//Check Error during FB_Init
IF THIS^.bErrorDuringFbInit THEN
	IF NOT fbInitError.bRaised THEN 
		//This error cannot be reset. Requires a reset cold
		fbInitError.CreateEx(stEventEntry:=TC_EVENTS.CHALET_Base_Events.ErrorFBinit, ipSourceInfo := THIS^.fbSourceInfo, bWithConfirmation := FALSE);
		fbInitError.Raise(0);
	END_IF
	Initialize:= E_FAIL;
	THIS^.fbFeedback.HR := Initialize;
	RETURN;
END_IF	

//Interface to System is missing
IF THIS^.ipXtsSystem = 0 THEN
	IF NOT fbMissingInterfaceAlarm.bRaised THEN 
		//This error cannot be reset. Requires a reset cold
		fbMissingInterfaceAlarm.CreateEx(stEventEntry:=TC_EVENTS.CHALET_XTS_Events.InitializationInvalideParameter, ipSourceInfo := THIS^.fbSourceInfo, bWithConfirmation := FALSE);
		fbMissingInterfaceAlarm.Raise(0);
	END_IF
	Initialize := E_FAIL;
	THIS^.fbFeedback.HR := Initialize;
	RETURN;
END_IF


IF NOT THIS^.bInitDone THEN
	
	THIS^.DeleteMoversQueue();

//	//Validate Settings - Error
//	bErrorStationInFrontNotFound := ((ipStationInFront = 0) AND THIS^.ipXtsSystem.Environment.TrackIsRing AND (THIS^.ipXtsSystem.Stations.Size > 1));
//	bErrorStationBehindeNotFound := ((ipStationBehinde = 0) AND THIS^.ipXtsSystem.Environment.TrackIsRing AND (THIS^.ipXtsSystem.Stations.Size > 1));		
//	IF (bErrorStationInFrontNotFound OR bErrorStationBehindeNotFound OR (THIS^.LUID = '') OR (fTrackLentgh <= 0) OR (fPositionOnTrack < 0.0) OR (fPositionOnTrack >= fTrackLentgh) OR (fMoverVelocityAtExit <= 0) OR (fMoverGapAtExit <= 0)) THEN
//		fbFeedback.hr := GetMostSignificant(E_FAIL, fbFeedback.hr);	
//		IF NOT fbInitError.bRaised THEN 
//			//This error cannot be reset. Requires a reset cold
//			fbInitError.CreateEx(stEventEntry:=TC_EVENTS.CHALET_XTS_Events.InitializationInvalideParameter, ipSourceInfo := THIS^.fbSourceInfo, bWithConfirmation := FALSE);
//			fbInitError.Raise(0);
//		END_IF
//	END_IF

		THIS^.fbTrigger.ListOfMoversToCheck := THIS^.ipXtsSystem.Movers;
		THIS^.fbTrigger.PositionOnTrack := THIS^.PositionOnTrack;
		THIS^.fbTrigger.TriggerDirection := MC_Positive_Direction;
		fbSortedListMoversInQueue.EndPositionOnTrack := LMOD(lr_Value:=(THIS^.PositionOnTrack + 10.0), lr_Arg:= THIS^.fTrackLentgh); 
		fbSortedListMoversInQueue.StartPositionOnTrack := LMOD(lr_Value:=(fbSortedListMoversInQueue.EndPositionOnTrack  + 0.0001), lr_Arg:= THIS^.fTrackLentgh); 
		fbSortedListMoversInQueue.ListOfMoversToCheck := THIS^.fbAssignedMovers;	
	bInitDone := TRUE;
END_IF

IF 	bInitDone THEN
	fbFeedback.hr := S_OK;	
END_IF
							
Initialize := fbFeedback.hr;
END_METHOD

{attribute 'monitoring':='call'}
//[mm] Every mover that leaves or passes the station gets this new gap as a target.
PROPERTY MoverGapAtExit : LREAL
GET
MoverGapAtExit := fMoverGapAtExit;
END_GET
SET
fMoverGapAtExit := MoverGapAtExit;
END_SET
END_PROPERTY

{attribute 'monitoring':='call'}
PROPERTY MoverPerMin : LREAL
GET
MoverPerMin := THIS^.fMoverPerMin;
END_GET
END_PROPERTY

{attribute 'monitoring':='call'}
PROPERTY MoverQueueSize : UINT
GET
MoverQueueSize := THIS^.nMoverQueueSize;
END_GET
SET
THIS^.nMoverQueueSize := MoverQueueSize;
END_SET
END_PROPERTY

{attribute 'monitoring':='call'}
PROPERTY MoversInPlace : BOOL
GET
THIS^.Prepare();//Prepare time-critical information, if not already done


MoversInPlace := bMoversInPlace;
END_GET
END_PROPERTY

{attribute 'monitoring':='call'}
PROPERTY MoversInQueue : REFERENCE TO ARRAY [0..(XtsParameterlist.MAX_MOVER_PER_SYSTEM-1)] OF I_XTS_Mover_PLC // Return a sorted list of movers in this zone. Index 0 is the mover in Front.
GET
MoversInQueue REF= THIS^.fbSortedListMoversInQueue.MoversInZone;
END_GET
END_PROPERTY

{attribute 'monitoring':='call'}
PROPERTY MoverVelocityAtExit : LREAL //[mm/s] Every mover that leaves or passes the station gets this new velocity as a target.
GET
MoverVelocityAtExit := fMoverVelocityAtExit;
END_GET
SET
fMoverVelocityAtExit := MoverVelocityAtExit;
END_SET
END_PROPERTY

PROPERTY OID : OTCID
GET
OID := THIS^.OIDStationInfo;
END_GET
END_PROPERTY

{attribute 'monitoring':='call'}
//[mm] from the beginning of the assigned track
PROPERTY PositionOnTrack : LREAL
GET
PositionOnTrack := fPositionOnTrack;
END_GET
SET
THIS^.ChangePos(PositionOnTrack);
END_SET
END_PROPERTY

(* 
	Use this Methode to calculate time sensitive date once each cycle. Example: read analog input and convert before do get Signal propertie
*)
METHOD PROTECTED Prepare : HRESULT
VAR_INST
	{attribute 'hide'}	
	nLastUpdatedCycleCount : UDINT;
END_VAR

VAR
	nLoopIndex : UINT;
	fExpectedDistanceToParent : LREAL;
	fPositionDifference : LREAL;
	nCycleTime_ms : UDINT;
	bMoverInQueue : BOOL;
	bTempMoverInPosition : BOOL;
	bTempMoverVeloZero : BOOL;
	bTempMoverInMonitoringTime : BOOL;
	bTempMoverThisStationAsTarged : BOOL;
END_VAR
VAR_INST
	{attribute 'hide'}
	nCycleCountInPos : UDINT;
END_VAR
//Check if this Cycle the dates are allready prepared. This is important for time sensitive informations.
IF nLastUpdatedCycleCount <> TwinCAT_SystemInfoVarList._TaskInfo[THIS^.TaskIndex].CycleCount THEN
	nLastUpdatedCycleCount := TwinCAT_SystemInfoVarList._TaskInfo[THIS^.TaskIndex].CycleCount ;


	(* Check if mover is in place. Time and Position window *)
	//If queuesize is zero, mover is never in place.
	IF nMoverQueueSize = 0 OR NOT ipXtsSystem.Enabled THEN
		THIS^.bMoversInPlace := FALSE;
		nCycleCountInPos := 0;
	ELSE
		//Get this task cycle Count and time 
		nCycleTime_ms := TwinCAT_SystemInfoVarList._TaskInfo[THIS^.nTaskIndex].CycleTime(*100ns*) / 10_000 ;
		
		bTempMoverInPosition := TRUE; bTempMoverVeloZero := TRUE; bTempMoverThisStationAsTarged := TRUE;
		fExpectedDistanceToParent := 0;
		FOR nLoopIndex := 0 TO (THIS^.nMoverQueueSize-1) DO
			IF THIS^.fbSortedListMoversInQueue.MoversInZone[nLoopIndex] <> 0 THEN
				//Check position and Gap - 1 mover do not have a gap
				IF nLoopIndex <> 0 THEN
					fExpectedDistanceToParent := fExpectedDistanceToParent + THIS^.fbSortedListMoversInQueue.MoversInZone[nLoopIndex].LastCmdTargedGap;
				END_IF
				bMoverInQueue		:= TRUE;
				
				fPositionDifference := F_GetDistToPosModulo(fTargedPosition := (THIS^.PositionOnTrack - fExpectedDistanceToParent),  fActualPosition :=  THIS^.fbSortedListMoversInQueue.MoversInZone[nLoopIndex].FullAccess.getAxisRef.NcToPlc.ModuloActPos, fModulo := THIS^.ipXtsSystem.TrackLength);
				IF fPositionDifference > (THIS^.ipXtsSystem.TrackLength/2) THEN
					fPositionDifference := (THIS^.ipXtsSystem.TrackLength - fPositionDifference);
				END_IF
				
				bTempMoverInPosition := bTempMoverInPosition AND (ABS(fPositionDifference) <= fTargetPosWindow );
				bTempMoverVeloZero := bTempMoverVeloZero AND (THIS^.fbSortedListMoversInQueue.MoversInZone[nLoopIndex].SetVelocity = 0);
				bTempMoverThisStationAsTarged := bTempMoverThisStationAsTarged AND ((THIS^.fbSortedListMoversInQueue.MoversInZone[nLoopIndex].TargedStation = THIS^.LUID));
			ELSE
				//Missing mover in queue
				bMoverInQueue := FALSE;
				EXIT;
			END_IF
		END_FOR
			
		//start time if mover position is ok
		IF bTempMoverInPosition  THEN
			nCycleCountInPos := nCycleCountInPos + 1;
		ELSE
			nCycleCountInPos := 0;
		END_IF
		
		bTempMoverInMonitoringTime := (UDINT_TO_TIME(nCycleCountInPos * nCycleTime_ms) >= tTargetPosMonitoringTime);
				
		THIS^.bMoversInPlace := bMoverInQueue AND bTempMoverInPosition AND bTempMoverInMonitoringTime AND bTempMoverThisStationAsTarged;// AND bTempMoverVeloZero;
	END_IF
	
	
END_IF
END_METHOD

{attribute 'monitoring':='call'}
PROPERTY ProcessSimulationActive : BOOL
GET
ProcessSimulationActive := THIS^.fSimulationProcessDuration > 0;
END_GET
END_PROPERTY

{attribute 'monitoring':='call'}
//prevent further movers from entering the station, 
//e.g. to prevent a collision. All movers that are already moving to reach this station will be stopped with a stop 
//and restarted with Ready True.
PROPERTY ReadyToRecvMovers : BOOL
GET
ReadyToRecvMovers := bReadyToRecvMovers;
END_GET
SET
VAR
	ipTempMover : I_XTS_Mover;
END_VAR
//Change to Not Ready:
IF (ReadyToRecvMovers = FALSE) AND (bReadyToRecvMovers <> ReadyToRecvMovers) THEN
	//halt all movers on the way
	fbAssignedMovers.ResetIterator();
	WHILE fbAssignedMovers.HasNextObject() DO
		IF ToMover(fbAssignedMovers.GetNextObject(),ipTempMover) THEN
			ipTempMover.HaltCA();	
		END_IF	
	END_WHILE
END_IF

//Change to Ready:
IF (ReadyToRecvMovers = TRUE) AND (bReadyToRecvMovers <> ReadyToRecvMovers) THEN
	//all movers that are on the way have probably been stopped before. when reactivated, the last move command is sent again.
	fbAssignedMovers.ResetIterator();
	WHILE fbAssignedMovers.HasNextObject() DO
		IF ToMover(fbAssignedMovers.GetNextObject(),ipTempMover) THEN
			ipTempMover.MoveAbsCA(	fPosition	:= THIS^.PositionOnTrack, 
								fVelocity 	:= ipTempMover.LastCmdTargedVelocity,  
								fGap 		:= ipTempMover.LastCmdTargedGap,  
								eDirection 	:= Tc3_Mc3Definitions.MC_DIRECTION.mcDirectionPositive);	
		END_IF	
	END_WHILE
END_IF

//Store new status
bReadyToRecvMovers := ReadyToRecvMovers;
END_SET
END_PROPERTY

METHOD SendMoversToStation : HRESULT //Send all Queued movers away by changing the targed station destination
VAR_INPUT
	sTargedStation	: STRING;
END_VAR
VAR
	nLoopIndex 		: UINT;;
	ipMover	: I_XTS_Mover;
END_VAR
//Invalide targed
IF sTargedStation = '' THEN
	SendMoversToStation := E_FAIL;
	RETURN;
END_IF

//Movers have not reached station and can not send away until complet
IF NOT THIS^.MoversInPlace THEN
	SendMoversToStation := E_FAIL;
	RETURN;
END_IF

//Send all Queued movers away by changing the targed station destination
FOR nLoopIndex := 0 TO nMoverQueueSize-1 DO
	IF THIS^.MoversInQueue[nLoopIndex] <> 0 AND_THEN __QUERYINTERFACE(THIS^.MoversInQueue[nLoopIndex],ipMover) THEN
		ipMover.TargedStation := sTargedStation;		
	END_IF
END_FOR
END_METHOD

//If a valid time (>0seconds) is set and the configured destination station exists, then the movers will be sent away automatically after this time from now on.
METHOD SimulationStart : HRESULT
VAR_INPUT
	fProcessDuration 	: LREAL; //[s]
	sTargedStation		: STRING; //LUID of the targed station to automatic send after the duration
END_VAR
VAR
	ipStation	: I_CH_Object;
	bValideLUID : BOOL;
END_VAR
//Search LUID in Stationslist
ipStation := THIS^.ipXtsSystem.Stations.FindLUID(sTargedStation);
bValideLUID := (ipStation <> 0); 

IF (fProcessDuration > 0) AND bValideLUID THEN
	//Valide config
	THIS^.fSimulationProcessDuration 	:=	fProcessDuration;
	THIS^.sSimulationTargedStation 		:=	sTargedStation;
	SimulationStart := S_OK;
ELSE
	//Simulation disabled
	THIS^.SimulationStop();
	SimulationStart := S_FALSE;
END_IF
END_METHOD

//If a valid time (>0seconds) is set and the configured destination station exists, then the movers will be sent away automatically after this time from now on.
METHOD SimulationStartEx : HRESULT
VAR_INPUT
	fProcessDuration 		: LREAL; //[s]
	ipStation				: I_Xts_Station_PLC; //unique station to automatic send after the duration
END_VAR
IF ipStation <> 0 THEN
	SimulationStartEx := THIS^.SimulationStart(fProcessDuration := fProcessDuration, sTargedStation := ipStation.LUID);

ELSE
	SimulationStartEx := S_FALSE;
END_IF
END_METHOD

METHOD SimulationStop : HRESULT
//Simulation disabled
THIS^.fSimulationProcessDuration 	:=	0;
THIS^.sSimulationTargedStation 		:=	'';
END_METHOD

{attribute 'monitoring':='call'}
PROPERTY StationBehinde : I_XTS_Station
GET
StationBehinde := ipStationBehinde;
END_GET
END_PROPERTY

{attribute 'monitoring':='call'}
PROPERTY StationsAhead : I_XTS_Station
GET
StationsAhead := ipStationInFront;
END_GET
END_PROPERTY

{attribute 'monitoring':='call'}
PROPERTY SuppressDynamicsChange : BOOL // Suppress to change the dynamic(Gap+velocity) of passing movers. This is usefull in startup
GET
SuppressDynamicsChange := bSuppressDynamicsChange;
END_GET
SET
bSuppressDynamicsChange := SuppressDynamicsChange;
END_SET
END_PROPERTY

{attribute 'monitoring':='call'}
//A time that is waited as soon as the mover is in the station (including the monitoring window) before “MoversInPlace” is set. e.g. used to stabilize the workpiece
PROPERTY TargetPosMonitoringTime : TIME
GET
TargetPosMonitoringTime := tTargetPosMonitoringTime;
END_GET
SET
tTargetPosMonitoringTime := TargetPosMonitoringTime;
END_SET
END_PROPERTY

{attribute 'monitoring':='call'}
//How many mm before the mover reaches the position is “MoversInPlace” set for the process. 
//This distance can also be set very large (e.g. 100mm) for moving past without stopping.
PROPERTY TargetPosWindow : LREAL
GET
TargetPosWindow := fTargetPosWindow;
END_GET
SET
fTargetPosWindow := TargetPosWindow;
END_SET
END_PROPERTY

//This sequence tries to transfer the mover to the next station in the direction of travel and checks whether the next station has space for it. 
//If the next station is a "dummy" that only changes the dynamics of the passing mover, this station is skipped and the next station is searched one ahead.
//If the station is fully occupied, no action is taken and a new search can be made in the next cycle.
METHOD PROTECTED TrySendMoverToNextStation : HRESULT
VAR_INPUT
	ipMover	: I_XTS_Mover;
	fVelocity : LREAL;
	fGap : LREAL;
END_VAR
VAR
	bStationIsOnlyForDynamicChanges : BOOL;
	bStationIsFull					: BOOL;
	bStationHanMoreMoverThanAllowed : BOOL;
	bStationHasAFreePlaceInQueue 	: BOOL;
	bStationIsTheTarged				: BOOL;
	bStationIsNotReadyToRecvMovers	: BOOL;
	
	ipMoverObject 		: I_CH_Object;
	ipTempStation 		: I_XTS_Station;	
	ipTargedStation 	: I_XTS_Station;

	nXpuNo 				: UINT;
	iMoverNo 			: UINT;
	stCommand 			: ST_TcIoXtsMoverCommand;	
END_VAR
//Invalide interface
IF ipMover = 0 THEN
	TrySendMoverToNextStation := E_FAIL;
	RETURN;
END_IF

//Mover is not in this Station.
IF __QUERYINTERFACE(ipMover,ipMoverObject) AND_THEN NOT THIS^.fbAssignedMovers.ObjectInList(ipMoverObject) THEN
	TrySendMoverToNextStation := E_FAIL;
	RETURN;
END_IF

//Send to actual Station is not supported
IF ipMover.TargedStation = THIS^.LUID THEN
	TrySendMoverToNextStation := E_FAIL;
	RETURN;
END_IF


ipTempStation := (THIS^);
//This sequence tries to transfer the mover to the next station in the direction of travel and checks whether the next station has space for it. 
//If the next station is a "dummy" that only changes the dynamics of the passing mover, this station is skipped and the next station is searched one ahead.
//If the station is fully occupied, no action is taken and a new search can be made in the next cycle.
WHILE (ipTargedStation=0) DO
	
	//get next station in flow direction
	ipTempStation := ipTempStation.StationsAhead;

	//All Stations around the XTS tested, Station not Found
	IF ipTempStation.LUID = THIS^.LUID THEN
		TrySendMoverToNextStation := E_FAIL;
		RETURN;
	END_IF

	bStationHanMoreMoverThanAllowed := (ipTempStation.CtsMoversInQueue > ipTempStation.MoverQueueSize); //Maybe during statup if all movers are forced to station x.	
	bStationIsFull					:= (ipTempStation.CtsEmptySpaceInQueue = 0) AND NOT (ipTempStation.MoverQueueSize = 0);
	bStationHasAFreePlaceInQueue 	:= (ipTempStation.CtsEmptySpaceInQueue > 0);
	bStationIsOnlyForDynamicChanges := (ipTempStation.MoverQueueSize = 0);
	bStationIsTheTarged				:= (ipTempStation.LUID = ipMover.TargedStation);
	bStationIsNotReadyToRecvMovers	:= ( NOT ipTempStation.ReadyToRecvMovers); 
	
	IF bStationIsFull OR bStationHanMoreMoverThanAllowed OR bStationIsNotReadyToRecvMovers THEN
		//Next Station is a valide targed but is already full.  Exit WHILE loop and try again next time.
		EXIT;
	
	ELSIF bStationHasAFreePlaceInQueue THEN
		//Next station found. Send mover to it.
		ipTargedStation := ipTempStation;
	
	ELSIF bStationIsOnlyForDynamicChanges AND bStationIsTheTarged THEN
		//ERROR. The target position is a dynamic station and can not be reached.
		TrySendMoverToNextStation := E_FAIL;
		RETURN;
		
	ELSIF bStationIsOnlyForDynamicChanges THEN
		//Repead WHILE loop and search an station more in front.
		;
	END_IF 

END_WHILE


//Requested station was found, send movers to there if it has space.
IF ipTargedStation <> 0 THEN
	//Handover Mover
	THIS^.fbAssignedMovers.RemoveObject(ipMoverObject);
	ipTargedStation.AddMoverToQueue(ipMover);
	//Start Movement
	ipMover.MoveAbsCA(
		fPosition:= ipTargedStation.PositionOnTrack, 
		fVelocity:= fVelocity, 
		fGap:= fGap, 
		eDirection:= Tc3_Mc3Definitions.MC_DIRECTION.mcDirectionPositive);
		
	//build Log Command
	stCommand.sCommandType	:= 'leaving station';
	stCommand.sStation		:= ipTargedStation.LUID;
	stCommand.sText 		:= F_BuildLogString(fPos := ipTargedStation.PositionOnTrack, fVelocity := fVelocity, fGap := fGap);

	//get Xpu Number by AxisId
	nXpuNo := ipXtsSystem.Environment.UtilityEnvirement.GetXpuNumberByAxisId(ipMover.getAxisRef.NcToPlc.AxisId);
	//get Mover Number by AxisId
	iMoverNo := ipXtsSystem.Environment.UtilityEnvirement.XpuTcIo(nXpuNo).GetMoverNumberByAxisId(ipMover.getAxisRef.NcToPlc.AxisId);
	
	//write Log Command
	ipXtsSystem.Environment.UtilityEnvirement.XpuTcIo(nXpuNo).MoverTcIo(iMoverNo).AddCommand(stCommand);
	

	
	TrySendMoverToNextStation := S_OK;	
ELSE
	//No movemnt possible, try next cycle again		
	TrySendMoverToNextStation := S_FALSE;
END_IF
END_METHOD

METHOD Update : HRESULT
VAR
	ipMover : I_XTS_Mover;
	ipThisStation : I_XTS_Station;
	fDistToNextMover : LREAL;
	fGapRequired : LREAL;
	bGapIsEnough : BOOL; //distance is large enough to start next command
END_VAR
//Force to do init befor call update
IF NOT bInitDone THEN
	THIS^.Initialize();
	RETURN;
END_IF


// Process Simulation. All functionality packed into one method for easier overwriting
THIS^.UpdateSimulation();


// If enabled start station logic
IF THIS^.ipXtsSystem.Enabled THEN
	
	ipThisStation := (THIS^);
	//Detect mover who is passing the station whitout be in queue. Adjust to new Gap+Dynamics
	IF fbTrigger.MoverDetected AND fbTrigger.MoverAtTrigger<>0 AND NOT THIS^.bSuppressDynamicsChange THEN
		//Only if not in this queue
		IF fbTrigger.MoverAtTrigger.ParentStation <> ipThisStation THEN
			fbTrigger.MoverAtTrigger.MoveAbsCA(
				fPosition:= fbTrigger.MoverAtTrigger.LastCmdTargedPosition, 
				fVelocity:= THIS^.fMoverVelocityAtExit, 
				fGap:= THIS^.fMoverGapAtExit, 
				eDirection:= Tc3_Mc3Definitions.MC_DIRECTION.mcDirectionPositive);
		END_IF
	END_IF
	
	///distance is large enough to start next command
	//This is to prevent stationary movers from having to move backwards
	IF THIS^.MoversInQueue[0] <> 0 THEN
		fDistToNextMover := F_GetDistToPosModulo(fTargedPosition:= THIS^.MoversInQueue[0].FullAccess.NextMover.PositionOnTrack, fActualPosition:= THIS^.MoversInQueue[0].PositionOnTrack, THIS^.ipXtsSystem.TrackLength);
		fGapRequired := MAX(THIS^.MoversInQueue[0].FullAccess.LastCmdTargedGap, THIS^.MoversInQueue[0].FullAccess.NextMover.LastCmdTargedGap);
		bGapIsEnough := (fDistToNextMover >= fGapRequired);
	END_IF
	
	
	//Test if the first mover is in station and send him away, if the destination is not this station
	IF __QUERYINTERFACE(THIS^.MoversInQueue[0],ipMover) AND_THEN (ipMover.TargedStation <> THIS^.LUID) AND_THEN bGapIsEnough THEN
		//IF mover is standstill in current station, send him away whit the exitVelocity, else use the in mover stored velocity
		IF (THIS^.MoversInQueue[0].PositionOnTrack = THIS^.PositionOnTrack) THEN
			THIS^.TrySendMoverToNextStation(ipMover := ipMover, fVelocity := THIS^.fMoverVelocityAtExit, fGap := THIS^.fMoverGapAtExit);
		ELSE
			THIS^.TrySendMoverToNextStation(ipMover := ipMover, fVelocity := ipMover.LastCmdTargedVelocity, fGap := ipMover.LastCmdTargedGap);
		END_IF	
      
	END_IF
END_IF


// Utility InfoStation, used in XTS Viewer. All functionality packed into one method for easier overwriting
THIS^.UpdateUtilityStation();

// Calculate statistic values like Mover/min of this station. All functionality packed into one method for easier overwriting
THIS^.UpdateStatistic();
END_METHOD

METHOD PROTECTED UpdateSimulation : HRESULT
VAR_INST
	tonSimulationDelay : TON;
END_VAR
//Automatic send mover to next station in Simulation
//If a valid time (>0seconds) is set and the configured destination station exists, then the movers will be sent away automatically after this time from now on.
tonSimulationDelay.IN 	:= THIS^.ipXtsSystem.Enabled AND THIS^.MoversInPlace AND THIS^.ProcessSimulationActive;
tonSimulationDelay.PT	:= LREAL_TO_TIME(THIS^.fSimulationProcessDuration*1000.0);
tonSimulationDelay();
IF tonSimulationDelay.Q THEN
	THIS^.SendMoversToStation(sTargedStation := THIS^.sSimulationTargedStation);
END_IF
END_METHOD

METHOD PROTECTED UpdateStatistic : HRESULT
VAR
	nCycleTime_ns : UDINT;
END_VAR
VAR_INST
	tWaitForXTS, tWaitForProcess 	: LTIME;
	nMoverPassingStation			: UINT;
END_VAR
//Validate settings. STATISTIC_AVG_PERIOD must be >0
IF NOT TIME_TO_BOOL(XtsParameterlist.STATISTIC_AVG_PERIOD) THEN
	UpdateStatistic := E_FAIL;
	RETURN;
END_IF

//Get this task cycle time
nCycleTime_ns := TwinCAT_SystemInfoVarList._TaskInfo[THIS^.nTaskIndex].CycleTime(*100ns*) * 100;


//Depending on whether the station gives the start signal to the process or not, decide which of the two times should be incremented.
IF THIS^.MoversInPlace THEN
	tWaitForProcess := tWaitForProcess + UDINT_TO_LTIME(nCycleTime_ns);
ELSE
	tWaitForXTS 	:= tWaitForXTS + UDINT_TO_LTIME(nCycleTime_ns);
END_IF


//Check for mover who is passing the station
IF THIS^.fbTrigger.MoverDetected THEN
	nMoverPassingStation := nMoverPassingStation +1;
END_IF


//Once the period is reached. Evaluate and reset
IF (tWaitForProcess + tWaitForXTS) >= TIME_TO_LTIME(XtsParameterlist.STATISTIC_AVG_PERIOD) THEN
	
	//Calculate passing mover per minute
	THIS^.fMoverPerMin := TO_LREAL(nMoverPassingStation)*TIME_TO_LREAL(TIME#1M)/TIME_TO_LREAL(XtsParameterlist.STATISTIC_AVG_PERIOD);

	
	
	tWaitForProcess	:= LTIME#0NS;
	tWaitForXTS 	:= LTIME#0NS;
	nMoverPassingStation := 0;
END_IF
END_METHOD

METHOD PROTECTED UpdateUtilityStation : HRESULT //Utility InfoStation, used in XTS Viewer. All functionality packed into one method for easier overwriting
VAR
	aStopPositionsInfoStation : ARRAY[1..Tc3_XTS_Utility.TcIoXtsEnvironmentParameterList.MaxXtsStopPositionsPerStation] OF LREAL;
	//aPartIDs : ARRAY[1..Tc3_XTS_Utility.TcIoXtsEnvironmentParameterList.MaxXtsPartsPerXpu] OF OTCID;
	fLastStopPosition 		: LREAL;
	nLoopIndex 				: UINT;	
    ipMovers 				: CHALET_BaseComponents.I_CH_List;
	ipTempMover 			: I_XTS_Mover;
	nXpuNo 					: UINT;
	nMoverNo 				: UINT;
	pObject 				: ITComObject;
	sName 					: STRING;
END_VAR


VAR_INST

	nOldMoverQueueSize 		: UINT := CHALET_BaseComponents.GVL_Datatypes.cMaxUint;
	fOldPositionOnTrack 	: LREAL;
	anBias 					: ARRAY[1..2] OF INT;
	bInverted 				: BOOL;
END_VAR
//Validate inputs
IF THIS^.OIDStationInfo = 0 OR ipXtsSystem.Environment = 0 THEN
	RETURN;
END_IF	


// Initalize
IF NOT THIS^.bUtilityStationInitDone THEN
	//Get interface to utility station belongs to this station via OID
    FOR nLoopIndex := 1 TO ipXtsSystem.Environment.UtilityEnvirement.InfoServerTcIo(1).P_InfoStationCount DO
		IF 	ipXtsSystem.Environment.UtilityEnvirement.InfoServerTcIo(1).P_InfoStationOids[nLoopIndex] = THIS^.OIDStationInfo THEN
			THIS^.ipStationInfo := ipXtsSystem.Environment.UtilityEnvirement.InfoServerTcIo(1).InfoStationTcIo(nInfoStation:= nLoopIndex);
			EXIT;
		END_IF
	END_FOR	
	
	// calculate Position Offset
	IF THIS^.ipStationInfo <> 0 THEN			
		ipMovers := ipXtsSystem.Movers;
		ipMovers.ResetIterator();
		nLoopIndex := 0;	
		WHILE ipMovers.HasNextObject() DO
			nLoopIndex := nLoopIndex + 1;
			IF ToMover(ipMovers.GetNextObject(),ipTempMover) THEN
				//get Xpu Number by AxisId
				nXpuNo := ipXtsSystem.Environment.UtilityEnvirement.GetXpuNumberByAxisId(ipTempMover.getAxisRef.NcToPlc.AxisId);
				//get Mover Number by AxisId
				nMoverNo := ipXtsSystem.Environment.UtilityEnvirement.XpuTcIo(nXpuNo).GetMoverNumberByAxisId(ipTempMover.getAxisRef.NcToPlc.AxisId);
				//calculate Bias
				anBias[nLoopIndex] := LREAL_TO_INT(ipXtsSystem.Environment.UtilityEnvirement.XpuTcIo(nXpuNo).MoverTcIo(nMoverNo).GetPositionInfo().fPartPosition - ipTempMover.getAxisRef.NcToPlc.ModuloActPos);
				IF nLoopIndex = 2 THEN
					 EXIT;
				END_IF
			END_IF
		END_WHILE
		
		// Validate bias, check for inverted direction
		IF anBias[1] <> anBias[2] THEN
			bInverted := TRUE; 
			ipMovers.ResetIterator();
			nLoopIndex := 0;	
			WHILE ipMovers.HasNextObject() DO
				nLoopIndex := nLoopIndex + 1;
				IF ToMover(ipMovers.GetNextObject(),ipTempMover) THEN
					//get Xpu Number by AxisId
					nXpuNo := ipXtsSystem.Environment.UtilityEnvirement.GetXpuNumberByAxisId(ipTempMover.getAxisRef.NcToPlc.AxisId);
					//get Mover Number by AxisId
					nMoverNo := ipXtsSystem.Environment.UtilityEnvirement.XpuTcIo(nXpuNo).GetMoverNumberByAxisId(ipTempMover.getAxisRef.NcToPlc.AxisId);
					//calculate inverted Bias
					anBias[nLoopIndex] := LREAL_TO_INT(ipXtsSystem.TrackLength - ipXtsSystem.Environment.UtilityEnvirement.XpuTcIo(nXpuNo).MoverTcIo(nMoverNo).GetPositionInfo().fPartPosition - ipTempMover.getAxisRef.NcToPlc.ModuloActPos);
					IF nLoopIndex = 2 THEN
						 EXIT;
					END_IF
				END_IF	
			END_WHILE
		END_IF
		
		//Set unique station name
		FW_ObjMgr_GetObjectInstance(oid:= THIS^.OIDStationInfo , iid:= TC_GLOBAL_IID_LIST.IID_ITComObject, pipUnk:= ADR(pObject));
		IF pObject <> 0 THEN
			sName := THIS^.LUID;
			pObject.TcSetObjectName(ADR(sName));
			pObject.TcRelease();
		END_IF

	END_IF
	
	THIS^.bUtilityStationInitDone := TRUE;
	fOldPositionOnTrack := -1;
END_IF




// Update
// Configure/draw station in viewer on change
IF (THIS^.ipStationInfo <> 0) AND (THIS^.nMoverQueueSize <> nOldMoverQueueSize OR THIS^.fPositionOnTrack <> fOldPositionOnTrack) THEN	
	nOldMoverQueueSize := THIS^.nMoverQueueSize;
	fOldPositionOnTrack := THIS^.fPositionOnTrack;
	
	THIS^.ipStationInfo.SetPartObjectIds(ipXtsSystem.Environment.UtilityEnvirement.XpuTcIo(1).P_PartOids);
	THIS^.ipStationInfo.SetIsEnabled(TRUE);

	
	// Draw stop position if gap between mover, given by station behind, is set
	IF (StationBehinde <> 0) AND (THIS^.nMoverQueueSize > 0) AND THIS^.nMoverQueueSize <= 25 THEN
		//Clear array
		MEMSET(ADR(aStopPositionsInfoStation), SIZEOF(aStopPositionsInfoStation), 0);
		//Fill array
		FOR nLoopIndex := 1 TO THIS^.nMoverQueueSize DO
			fLastStopPosition := (nLoopIndex-1)*StationBehinde.MoverGapAtExit;
			aStopPositionsInfoStation[(nLoopIndex)] := (fLastStopPosition);
		END_FOR
		IF NOT bInverted THEN
			//Start Position
			THIS^.ipStationInfo.SetStartPositionOnPart(MAX((fPositionOnTrack + anBias[1] - fLastStopPosition), 0)); ///zzz Todo. The InfoStation can not draw stations in the modulo area
			//End Pos
			THIS^.ipStationInfo.SetEndPositionOnPart(fPositionOnTrack + anBias[1]);
		ELSE
			//Start Position
			THIS^.ipStationInfo.SetStartPositionOnPart(ipXtsSystem.TrackLength - (fPositionOnTrack + anBias[1]));					
			//End Pos
			THIS^.ipStationInfo.SetEndPositionOnPart(MAX((ipXtsSystem.TrackLength - (fPositionOnTrack + anBias[1] - fLastStopPosition)), 0)); ///zzz Todo. The InfoStation can not draw stations in the modulo area
		END_IF
		//StopPositions
		THIS^.ipStationInfo.SetStopPositions(aStopPositionsInfoStation);

		//Override color if is set to transparent
		IF THIS^.ipStationInfo.GetStationColor() = 0 THEN
			THIS^.ipStationInfo.SetStationColor(nStationColor:= CHALET_BaseComponents.E_Colors_ARGB.Darkred);
		END_IF
	ELSE
		//Clear array
		MEMSET(ADR(aStopPositionsInfoStation), SIZEOF(aStopPositionsInfoStation), 0);	
		//StopPositions
		THIS^.ipStationInfo.SetStopPositions(aStopPositionsInfoStation);
		//Start Pos
		THIS^.ipStationInfo.SetStartPositionOnPart(nStartPositionOnPart := fPositionOnTrack + anBias[1]);
		//End Position
		THIS^.ipStationInfo.SetEndPositionOnPart(nEndPositionOnPart := fPositionOnTrack + anBias[1]);
	END_IF
	
	
	
	//Color Station depending on function:
	// Waitingstation green
	IF (FIND(THIS^.LUID,'wait')>0) OR (FIND(THIS^.LUID,'Wait')>0) OR (FIND(THIS^.LUID,'Warte')>0) OR (FIND(THIS^.LUID,'warte')>0) THEN
		THIS^.UtilityStationInfo.SetStationColor(nStationColor := CHALET_BaseComponents.E_Colors_ARGB.Green);
	
	// Dynamicstation blue
	ELSIF THIS^.MoverQueueSize = 0 THEN
		THIS^.UtilityStationInfo.SetStationColor(nStationColor := CHALET_BaseComponents.E_Colors_ARGB.Royalblue);	
    
	// Process station red
	ELSE
		THIS^.UtilityStationInfo.SetStationColor(nStationColor := CHALET_BaseComponents.E_Colors_ARGB.Red);			
	END_IF

END_IF
END_METHOD

{attribute 'monitoring':='call'}
PROPERTY UtilityStationInfo : I_TcIoXtsInfoServerInfoStation
GET
UtilityStationInfo := THIS^.ipStationInfo;
END_GET
END_PROPERTY

END_FUNCTION_BLOCK

// ---- COMPENENTs/Trigger/FB_XTS_Trigger.TcPOU
{attribute 'no_explicit_call' := 'Do not call the body - Stick to OOP'}
FUNCTION_BLOCK FB_XTS_Trigger EXTENDS FB_CH_Object IMPLEMENTS I_XTS_Trigger
VAR
	{attribute 'hide'}
	bInitDone : BOOL;
	{attribute 'hide'}
	ipXtsSystem : I_XTS_System_Registration;
	{attribute 'hide'}
	ipListOfMoversToCheck : CHALET_BaseComponents.I_CH_LIST;
	{attribute 'hide'}
	fTriggerPositionOnTrack : LREAL;
	{attribute 'hide'}
	eTriggerDirection : Tc2_MC2.MC_Direction := MC_Positive_Direction;
	{attribute 'hide'}
	ipMoverAtTrigger : I_XTS_Mover;
	{attribute 'hide'}	
	fTrackLentgh : LREAL;
	{attribute 'hide'}
	aMoversPositionLastCycle : ARRAY [0..(XtsParameterlist.MAX_MOVER_PER_SYSTEM-1)] OF LREAL; // This list is generated at the end of the PRG and contais the positions. The positions are checked in the next cycle
	{attribute 'hide'}
	aMoversInterfaceLastCycle : ARRAY [0..(XtsParameterlist.MAX_MOVER_PER_SYSTEM-1)] OF I_XTS_Mover; // This list is generated at the end of the PRG and contais the Mover interface. The positions are checked in the next cycle
	
END_VAR

METHOD FB_init : BOOL
VAR_INPUT
	bInitRetains : BOOL; // if TRUE, the retain variables are initialized (warm start / cold start)
	bInCopyCode : BOOL;  // if TRUE, the instance afterwards gets moved into the copy code (online change)
	
	ipXtsSystem : I_XTS_System_Registration; //Interface to XTS system object
	
END_VAR
VAR_INST
	{attribute 'hide'}
	bFBInitCalledOnce : BOOL; //Do the following code once during start up and not during onlinechange
END_VAR
//Do the following code once during start up and not during onlinechange
IF NOT bFBInitCalledOnce THEN 
	;
END_IF

//Regristrate object in System if unknown
IF ipXtsSystem <> 0 AND THIS^.ipXtsSystem = 0 THEN
	ipXtsSystem.RegisterTrigger(THIS^);
	THIS^.ipXtsSystem := ipXtsSystem;
END_IF

bFBInitCalledOnce := TRUE;
END_METHOD

{attribute 'monitoring':='call'}
PROPERTY HR : HRESULT
GET
///zzz todo
END_GET
END_PROPERTY

METHOD Initialize : HRESULT
IF THIS^.ipXtsSystem = 0 THEN
	//No valide interface
	Initialize := E_FAIL;
	RETURN;
END_IF

//Store track information
THIS^.fTrackLentgh := THIS^.ipXtsSystem.TrackLength;

IF (THIS^.ipListOfMoversToCheck <> 0) AND (THIS^.fTrackLentgh > 0.0) THEN
	THIS^.bInitDone := TRUE;
	Initialize := S_OK;
ELSE
	Initialize := E_FAIL;
END_IF
END_METHOD

PROPERTY ListOfMoversToCheck : I_CH_List
SET
IF ListOfMoversToCheck <> 0 THEN
	ipListOfMoversToCheck := ListOfMoversToCheck;
END_IF
END_SET
END_PROPERTY

{attribute 'monitoring':='call'}
PROPERTY MoverAtTrigger : I_XTS_Mover
GET
THIS^.Prepare();//Prepare Time-critical information

MoverAtTrigger := ipMoverAtTrigger;
END_GET
END_PROPERTY

{attribute 'monitoring':='call'}
PROPERTY MoverDetected : BOOL
GET
THIS^.Prepare();//Prepare Time-critical information

MoverDetected := (ipMoverAtTrigger <> 0);
END_GET
END_PROPERTY

{attribute 'monitoring':='call'}
PROPERTY PositionOnTrack : LREAL
GET
PositionOnTrack := fTriggerPositionOnTrack;
END_GET
SET
fTriggerPositionOnTrack := PositionOnTrack;
END_SET
END_PROPERTY

(* Time-critical information is processed here, which can then be polled via the property every cycle. 
The update method is usually at the end of the program and then it is already 'outdated'. *)
METHOD PRIVATE Prepare : HRESULT
VAR
	fMoverActPos,fMoverLastPos : LREAL;
	fRangePositive, fRangeNegative : LREAL;
	bMoverWasInRangeNeg, bMoverWasInRangePos, bMoverIsInRangeNeg, bMoverIsInRangePos : BOOL;
	nLoopIndex : UINT;
END_VAR
VAR_INST
	{attribute 'hide'}
	nLastUpdatedCycleCount : UDINT;
END_VAR
VAR CONSTANT
	cMaxMoveDistPerCycle : LREAL := 4000.0 * 20.0 / 1000.0 * 1.1; //4 m/s(max. XTS speed) * 20ms(max realistic SPS cycle time) + 10%
END_VAR
//Check if this Cycle the dates are allready prepared
IF nLastUpdatedCycleCount <> TwinCAT_SystemInfoVarList._TaskInfo[THIS^.nTaskIndex].CycleCount THEN
	nLastUpdatedCycleCount := TwinCAT_SystemInfoVarList._TaskInfo[THIS^.nTaskIndex].CycleCount;

	//Clear last stored Mover if an new cycle has started
	THIS^.ipMoverAtTrigger := 0;
	
	//Check old list of Moverspositions and compare them to the current position of the same mover.
	//Set Trigger if the Mover pass the Station
	fRangePositive := LMOD(lr_Value:=(THIS^.fTriggerPositionOnTrack + cMaxMoveDistPerCycle + THIS^.fTrackLentgh),lr_Arg:= THIS^.fTrackLentgh);
	fRangeNegative := LMOD(lr_Value:=(THIS^.fTriggerPositionOnTrack - cMaxMoveDistPerCycle + THIS^.fTrackLentgh),lr_Arg:= THIS^.fTrackLentgh);
	
	FOR nLoopIndex := 0 TO (XtsParameterlist.MAX_MOVER_PER_SYSTEM-1) DO
		IF aMoversInterfaceLastCycle[nLoopIndex] <> 0 THEN
			fMoverActPos :=  aMoversInterfaceLastCycle[nLoopIndex].PositionOnTrack;
			fMoverLastPos:=  aMoversPositionLastCycle[nLoopIndex];
			
			
			//Test if the the Mover was in Trigger-100mm Range(without exact the trigger point) and is now in Trigger+100 Range(with exact the trigger point)
			bMoverWasInRangePos	:= F_InLimitTest(fMinimum :=THIS^.fTriggerPositionOnTrack, fInput:= fMoverLastPos, fMaximum:=fRangePositive) AND NOT (fMoverLastPos=THIS^.fTriggerPositionOnTrack); 
			bMoverWasInRangeNeg	:= F_InLimitTest(fMinimum :=fRangeNegative, fInput:= fMoverLastPos, fMaximum:=THIS^.fTriggerPositionOnTrack) AND NOT (fMoverLastPos=THIS^.fTriggerPositionOnTrack); 
			bMoverIsInRangePos 	:= F_InLimitTest(fMinimum :=THIS^.fTriggerPositionOnTrack, fInput:= fMoverActPos, fMaximum:=fRangePositive); 
			bMoverIsInRangeNeg 	:= F_InLimitTest(fMinimum :=fRangeNegative, fInput:= fMoverActPos, fMaximum:=THIS^.fTriggerPositionOnTrack); 
		
			IF eTriggerDirection = MC_Positive_Direction AND bMoverWasInRangeNeg AND bMoverIsInRangePos THEN
				THIS^.ipMoverAtTrigger := aMoversInterfaceLastCycle[nLoopIndex];
				RETURN;
			ELSIF eTriggerDirection = MC_Negative_Direction AND bMoverIsInRangeNeg AND bMoverWasInRangePos THEN
				THIS^.ipMoverAtTrigger := aMoversInterfaceLastCycle[nLoopIndex];
				RETURN;	
			END_IF
			
		END_IF
	END_FOR
END_IF
END_METHOD

{attribute 'monitoring':='call'}
PROPERTY TimeStamp : Tc2_EtherCAT.T_DCTIME64
GET
THIS^.Prepare();//Prepare Time-critical information

///zzz todo exact time stamp calculatioin
 IF ipMoverAtTrigger <> 0 THEN
	 TimeStamp := F_GetCurDcTaskTime64();
 ELSE
	 TimeStamp := 0;
 END_IF
END_GET
END_PROPERTY

{attribute 'monitoring':='call'}
PROPERTY TriggerDirection : Tc2_MC2.MC_Direction
GET
TriggerDirection := eTriggerDirection;
END_GET
SET
IF TriggerDirection = MC_Positive_Direction OR TriggerDirection = MC_Negative_Direction THEN
	eTriggerDirection := TriggerDirection;
END_IF
END_SET
END_PROPERTY

METHOD Update : HRESULT
VAR
	nIndex : UINT;
	ipMover : I_XTS_Mover;
END_VAR
//Force to do an init befor call update
IF NOT bInitDone THEN
	THIS^.Initialize();
	RETURN;
END_IF

//Clear array
MEMSET(destAddr:=ADR(aMoversInterfaceLastCycle),n:=SIZEOF(aMoversInterfaceLastCycle),fillByte:=0);
MEMSET(destAddr:=ADR(aMoversPositionLastCycle),n:=SIZEOF(aMoversPositionLastCycle),fillByte:=0);

nIndex := 0;
THIS^.ipListOfMoversToCheck.ResetIterator();
WHILE THIS^.ipListOfMoversToCheck.HasNextObject() DO
	
	//Cheack all Movers fill the actposition in the array
	IF ToMover(THIS^.ipListOfMoversToCheck.GetNextObject(),ipMover) THEN
		aMoversInterfaceLastCycle[nIndex] := ipMover;
		aMoversPositionLastCycle[nIndex] := ipMover.PositionOnTrack;
		nIndex := nIndex +1;
	END_IF
	
END_WHILE
END_METHOD

END_FUNCTION_BLOCK

// ---- FUNCTIONs/F_InLimitTest.TcPOU
FUNCTION F_InLimitTest : BOOL
VAR_INPUT
	fMinimum 	: LREAL;
	fMaximum 	: LREAL;
	fInput 		: LREAL;
END_VAR

//Normal case
// 9 Max
// 5 Test
// 1 Min
IF fMinimum <= fMaximum THEN
	F_InLimitTest := (fInput >= fMinimum) AND (fInput <= fMaximum);
	
//Modulo case	
// 6 | 6  Max
// 5 | 9  Test
// 8 | 8  Min
ELSIF fMinimum > fMaximum THEN
	F_InLimitTest := NOT((fInput > fMaximum) AND (fInput < fMinimum));
END_IF

END_FUNCTION

// ---- COMPENENTs/Zone/FB_XTS_Zone.TcPOU
{attribute 'no_explicit_call' := 'Do not call the body - Stick to OOP'}
// Check zone start to end in positive direktion.
FUNCTION_BLOCK FB_XTS_Zone EXTENDS FB_CH_Object IMPLEMENTS I_XTS_Zone
VAR
	{attribute 'hide'}
	bInitDone : BOOL;
	{attribute 'hide'}
	ipXtsSystem : I_XTS_System_Registration;
	
	{attribute 'hide'}
	ipListOfMoversToCheck : CHALET_BaseComponents.I_CH_LIST;
	{attribute 'hide'}
	aMoversInZone : ARRAY [0..(XtsParameterlist.MAX_MOVER_PER_SYSTEM-1)] OF I_XTS_Mover_PLC;
	{attribute 'hide'}
	fStartPositionOnTrack : LREAL;
	{attribute 'hide'}
	fEndPositionOnTrack : LREAL;	
	{attribute 'hide'}
	fTrackLentgh : LREAL;
END_VAR

{attribute 'monitoring':='call'}
PROPERTY CtsMoversInZone : UINT
GET
VAR
	nIndex : UINT;
END_VAR
THIS^.Prepare();//Prepare Time-critical information

//Check array for entrys, exit if fisrt empty arrayindex is found.
FOR nIndex := 0 TO (XtsParameterlist.MAX_MOVER_PER_SYSTEM-1) DO
	IF (aMoversInZone[nIndex] <> 0) THEN
		CtsMoversInZone := CtsMoversInZone +1;
	ELSE
		RETURN;
	END_IF
END_FOR
END_GET
END_PROPERTY

{attribute 'monitoring':='call'}
PROPERTY EndPositionOnTrack : LREAL
GET
EndPositionOnTrack := fEndPositionOnTrack;
END_GET
SET
fEndPositionOnTrack := EndPositionOnTrack;
END_SET
END_PROPERTY

METHOD FB_init : BOOL
VAR_INPUT
	bInitRetains : BOOL; // if TRUE, the retain variables are initialized (warm start / cold start)
	bInCopyCode : BOOL;  // if TRUE, the instance afterwards gets moved into the copy code (online change)
	
	ipXtsSystem : I_XTS_System_Registration; //Interface to XTS system object
END_VAR
VAR_INST
	{attribute 'hide'}
	bFBInitCalledOnce : BOOL; //Do the following code once during start up and not during onlinechange
END_VAR
//Do the following code once during start up and not during onlinechange
IF NOT bFBInitCalledOnce THEN 
	;
END_IF

//Regristrate object in System if unknown
IF ipXtsSystem <> 0 AND THIS^.ipXtsSystem = 0 THEN
	ipXtsSystem.RegisterZone(THIS^);
	THIS^.ipXtsSystem := ipXtsSystem;
END_IF

bFBInitCalledOnce := TRUE;
END_METHOD

{attribute 'monitoring':='call'}
PROPERTY HR : HRESULT
GET
IF CHALET_BaseComponents.BaseParameterlist.MAX_OBJECTS > XtsParameterlist.MAX_MOVER_PER_SYSTEM THEN
	HR := E_FAIL;
END_IF
END_GET
END_PROPERTY

METHOD Initialize : HRESULT
IF THIS^.ipXtsSystem = 0 THEN
	//No valide interface
	Initialize := E_FAIL;
	RETURN;
END_IF

//Store track information
THIS^.fTrackLentgh := THIS^.ipXtsSystem.TrackLength;

IF (THIS^.ipListOfMoversToCheck <> 0) AND (THIS^.fTrackLentgh > 0.0) THEN
	THIS^.bInitDone := TRUE;
	Initialize := S_OK;
ELSE
	Initialize := E_FAIL;
END_IF
END_METHOD

PROPERTY ListOfMoversToCheck : I_CH_List
SET
IF ListOfMoversToCheck <> 0 THEN
	ipListOfMoversToCheck := ListOfMoversToCheck;
END_IF
END_SET
END_PROPERTY

{attribute 'monitoring':='call'}
PROPERTY MoversInZone : REFERENCE TO ARRAY [0..(XtsParameterlist.MAX_MOVER_PER_SYSTEM-1)] OF I_XTS_Mover_PLC // Return a sorted list of movers in this zone. Index 0 is the mover in Front.
GET
THIS^.Prepare();//Prepare Time-critical information

MoversInZone REF= THIS^.aMoversInZone;
END_GET
END_PROPERTY

(* Time-critical information is processed here, which can then be polled via the property every cycle. 
The update method is usually at the end of the program and then it is already 'outdated'. *)
METHOD PRIVATE Prepare : HRESULT
VAR
	nLoopIndex : UINT;
	ipMoverPlc : I_XTS_Mover_PLC;
	fDistToStart : LREAL;
	aDisanceToStart : ARRAY [0..XtsParameterlist.MAX_MOVER_PER_SYSTEM] OF LREAL;
END_VAR
VAR_INST
	{attribute 'hide'}
	nLastUpdatedCycleCount : UDINT;
END_VAR
//Check if this Cycle the dates are allready prepared
IF nLastUpdatedCycleCount <> TwinCAT_SystemInfoVarList._TaskInfo[THIS^.nTaskIndex].CycleCount THEN
	nLastUpdatedCycleCount := TwinCAT_SystemInfoVarList._TaskInfo[THIS^.nTaskIndex].CycleCount;

	//Clear array
	MEMSET(destAddr:=ADR(aMoversInZone),n:=SIZEOF(aMoversInZone),fillByte:=0);
	
	//Cheack all Movers and generate a sorted list of all mover in this zone
	THIS^.ipListOfMoversToCheck.ResetIterator();
	WHILE THIS^.ipListOfMoversToCheck.HasNextObject() DO
		IF ToMover_PLC(THIS^.ipListOfMoversToCheck.GetNextObject(),ipMoverPlc) THEN
			
			//If in zone
			IF F_InLimitTest(fMinimum:= fStartPositionOnTrack, fMaximum:=fEndPositionOnTrack, fInput:= ipMoverPlc.PositionOnTrack) THEN
				fDistToStart := F_GetDistToPosModulo(fActualPosition:= ipMoverPlc.PositionOnTrack, fTargedPosition:= fEndPositionOnTrack, fModulo := fTrackLentgh);
				
				//Check array of movers and decide if the current one is closer to 
				FOR nLoopIndex := 0 TO (XtsParameterlist.MAX_MOVER_PER_SYSTEM-1) DO
					//empty array position
					IF aMoversInZone[nLoopIndex] = 0 THEN
						aMoversInZone[nLoopIndex] := ipMoverPlc;
						aDisanceToStart[nLoopIndex] := fDistToStart;
						EXIT;
						
					//Closer Mover found, move whole array 	
					ELSIF aDisanceToStart[nLoopIndex] > fDistToStart THEN
						MEMMOVE(srcAddr := ADR(aMoversInZone[nLoopIndex]), destAddr := ADR(aMoversInZone[nLoopIndex+1]), n := (SIZEOF(aMoversInZone[0])*(XtsParameterlist.MAX_MOVER_PER_SYSTEM-nLoopIndex-1)));
						MEMMOVE(srcAddr := ADR(aDisanceToStart[nLoopIndex]), destAddr := ADR(aDisanceToStart[nLoopIndex+1]), n := (SIZEOF(aDisanceToStart[0])*(XtsParameterlist.MAX_MOVER_PER_SYSTEM-nLoopIndex-1)));
						aMoversInZone[nLoopIndex] := ipMoverPlc;
						aDisanceToStart[nLoopIndex] := fDistToStart;
						EXIT;
						
					//check next position	
					ELSE 
						;
					END_IF
				END_FOR
			END_IF
		END_IF
	END_WHILE
END_IF
END_METHOD

{attribute 'monitoring':='call'}
PROPERTY StartPositionOnTrack : LREAL
GET
StartPositionOnTrack := fStartPositionOnTrack;
END_GET
SET
fStartPositionOnTrack := StartPositionOnTrack;
END_SET
END_PROPERTY

METHOD Update : HRESULT
VAR

END_VAR
// Nothing todo in Update. Check Prepare
END_METHOD

END_FUNCTION_BLOCK

// ---- FUNCTIONs/F_GetDistToPosModulo.TcPOU
FUNCTION F_GetDistToPosModulo : LREAL //This is only working in Positiv Direktion
VAR_INPUT
	fTargedPosition : LREAL;
	fActualPosition : LREAL;
	fModulo 		: LREAL;
END_VAR

VAR

END_VAR

//Invalide input
IF fModulo = 0 THEN
	F_GetDistToPosModulo := 0;
	RETURN;
END_IF



//The MODABS function performs a modulo division and determines the unsigned modulo value within the modulo range.
	//Examples
	//MODABS(400.56, 360) = 40.56
	//MODABS(-400.56, 360) = 319.44
fTargedPosition := MODABS(fTargedPosition, fModulo);
fActualPosition := MODABS(fActualPosition, fModulo);
	
	
	
IF fTargedPosition < fActualPosition THEN
	fTargedPosition := fTargedPosition + fModulo;
END_IF

F_GetDistToPosModulo := fTargedPosition - fActualPosition;

END_FUNCTION

// ---- FUNCTIONs/F_BuildLogString.TcPOU
FUNCTION F_BuildLogString : String
VAR_INPUT
	fPos : LREAL;
	fVelocity : LREAL;
	fGap : LREAL;
END_VAR
VAR
	sTemp: STRING;
END_VAR

sTemp := 				CONCAT('Pos:' , LREAL_TO_STRING(fPos));
sTemp := CONCAT(sTemp, 	CONCAT(', Velocity:' , LREAL_TO_STRING(fVelocity)));
sTemp := CONCAT(sTemp, 	CONCAT(', Gap:' , LREAL_TO_STRING(fGap)));

F_BuildLogString := sTemp;

END_FUNCTION

// ---- COMPENENTs/System/FB_XTS_System.TcPOU
{attribute 'no_explicit_call' := 'Do not call the body - Stick to OOP'}
(* XTS System - 1 per associated XTS 
	The system is the container and organizer for all subsequent XTS objects. All objects are registered with this system*)
FUNCTION_BLOCK FB_XTS_System EXTENDS FB_CH_Object IMPLEMENTS I_XTS_System_Registration, I_XTS_System_PLC
VAR	
	{attribute 'hide'}
	bInitDone : BOOL;
	bErrorDuringFbInit : BOOL; // Not possible to reset
	{attribute 'hide'}                   	
	eActiveCommand 		: CHALET_Nc.E_NcAxisCommands := CHALET_Nc.E_NcAxisCommands.None;
	{attribute 'hide'}
    fbMovers     : CHALET_BaseComponents.FB_CH_List;
	{attribute 'hide'}	
	fbStations 	 : CHALET_BaseComponents.FB_CH_List;
	{attribute 'hide'}	
	fbZones 	 : CHALET_BaseComponents.FB_CH_List;
	{attribute 'hide'}	
	fbTriggers 	 : CHALET_BaseComponents.FB_CH_List;
	{attribute 'hide'}	
	ipGroup		 : I_XTS_Group;
	{attribute 'hide'}	
    ipEnvironment : I_XTS_Environment;
	{attribute 'hide'}
    nSeqEnabling  : UINT;
	{attribute 'hide'}	
    nSeqDisabling  : UINT;
	{attribute 'hide'}	
	fbFeedback : CHALET_BaseComponents.FB_CH_Feedback(ipSourceInfo := fbSourceInfo);
END_VAR
VAR CONSTANT
	{attribute 'hide'}
	SEQ_DONE : UINT := 999;
END_VAR

METHOD Disable : CHALET_BaseComponents.I_CH_Feedback
//prevent a mover from a station from getting a new position at high speed when stopped
THIS^.SuppressAllDynamicsChanges := TRUE;	

//Disable is allways posible

THIS^.nSeqDisabling 	:= 1;
THIS^.nSeqEnabling 		:= 0;

THIS^.eActiveCommand 				:= CHALET_NC.E_NcAxisCommands.Disable;
THIS^.fbFeedback.LastCommandAccepted:= TRUE;		
THIS^.fbFeedback.Busy 				:= TRUE;
		
Disable := THIS^.fbFeedback;
END_METHOD

{attribute 'monitoring':='call'}
PROPERTY Disabled : BOOL
GET
Disabled := nSeqDisabling = SEQ_DONE OR 
			(nSeqDisabling = 0 AND nSeqEnabling = 0);
END_GET
END_PROPERTY

METHOD PROTECTED Disabling : HRESULT
VAR
	hr : HRESULT;
	bOk : BOOL := TRUE;
	ipTempMover : I_XTS_Mover;
END_VAR

VAR_INST
	fbTimeWait : TON; 
	hrLastCycle : HRESULT;
END_VAR
Disabling := S_PENDING;
CASE nSeqDisabling OF
	0: // Idle
		Disabling := S_OK;
		
		
	1: // Halt movers
		THIS^.fbMovers.ResetIterator();
		WHILE THIS^.fbMovers.HasNextObject() DO
			IF ToMover(THIS^.fbMovers.GetNextObject(),ipTempMover) THEN
				IF ipTempMover.MoverInGroup AND NOT ipTempMover.getAxisRef.Status.HasBeenStopped THEN
					hr := GetMostSignificant(hr, ipTempMover.HaltCA());
				END_IF
			END_IF
		END_WHILE
		
		//Ignore feedback at this step. in next seq the movers get reseted.
		nSeqDisabling := 20;
		
	20: // Halting movers	
		THIS^.fbMovers.ResetIterator();
		WHILE THIS^.fbMovers.HasNextObject() DO
			IF ToMover(THIS^.fbMovers.GetNextObject(),ipTempMover) THEN
				bOk := bOk AND ipTempMover.getAxisRef.NcToPlc.SetVelo = 0;
			END_IF
		END_WHILE
		
		IF bOk THEN 
			nSeqDisabling := 25;
		END_IF	
		
		
	25: // wait for halt done
		IF THIS^.ipGroup.AllAxesStanding THEN
			nSeqDisabling := 30;
		END_IF
					
		
	30: // Reset movers
		THIS^.fbMovers.ResetIterator();
		WHILE THIS^.fbMovers.HasNextObject() DO
			IF ToMover(THIS^.fbMovers.GetNextObject(),ipTempMover) THEN
				hr := GetMostSignificant(hr, ipTempMover.Reset());
			END_IF
		END_WHILE
		
		IF CheckOk(hr) THEN 
			nSeqDisabling := 40;
		ELSE
			nSeqDisabling := 1000 + nSeqDisabling;
		END_IF				
		
		
	40: // Resetting movers
		THIS^.fbMovers.ResetIterator();
		WHILE THIS^.fbMovers.HasNextObject() DO
			IF ToMover(THIS^.fbMovers.GetNextObject(),ipTempMover) THEN
				hr := GetMostSignificant(hr, ipTempMover.Feedback.HR);
			END_IF
		END_WHILE
		
		IF CheckOk(hr) THEN 
			nSeqDisabling := 63;
		ELSIF FAILED(hr) THEN
			nSeqDisabling := 1000 + nSeqDisabling;
		END_IF
	
		
	63: // Reset group
		hr :=  THIS^.ipGroup.Reset();
		
		IF CheckOk(hr) THEN 
			nSeqDisabling := 64;
		ELSE
			nSeqDisabling := 1000 + nSeqDisabling;
		END_IF		
		
		
	64: // Resetting group
		hr := THIS^.ipGroup.HR;
		
		IF CheckOk(hr) THEN 
			nSeqDisabling := 70;
		ELSIF FAILED(hr) THEN
			nSeqDisabling := 1000 + nSeqDisabling;
		END_IF		
		
		
	70: // Disable group
		hr := THIS^.ipGroup.Disable();
		
		IF CheckOk(hr) THEN 
			nSeqDisabling := 100;
		ELSE
			nSeqDisabling := 1000 + nSeqDisabling;
		END_IF	
		
		
   100: // Disabling group
		hr := THIS^.ipGroup.HR;
		
		IF CheckOk(hr) THEN 
			nSeqDisabling := 110;
		ELSIF FAILED(hr) THEN
			nSeqDisabling := 1000 + nSeqDisabling;
		END_IF			
		
		
	110: // Remove movers from group
		hr := THIS^.ipGroup.UngroupAllAxes();
		
		IF CheckOk(hr) THEN 
			nSeqDisabling := 120;
		ELSE
			nSeqDisabling := 1000 + nSeqDisabling;
		END_IF		
	
		
	120: // Removing movers from group
		hr := THIS^.ipGroup.HR;
		
		IF CheckOk(hr) THEN 
			nSeqDisabling := 130;
		ELSIF FAILED(hr) THEN
			nSeqDisabling := 1000 + nSeqDisabling;
		END_IF	

		
	130: // write state to movers
		THIS^.fbMovers.ResetIterator();
		WHILE THIS^.fbMovers.HasNextObject() DO
			IF ToMover(THIS^.fbMovers.GetNextObject(),ipTempMover) THEN
				ipTempMover.MoverInGroup := FALSE;
			END_IF
		END_WHILE

		nSeqDisabling := 170;	
		
		
	170: // Disable movers
		THIS^.fbMovers.ResetIterator();
		WHILE THIS^.fbMovers.HasNextObject() DO
			IF ToMover(THIS^.fbMovers.GetNextObject(),ipTempMover) THEN
				hr := GetMostSignificant(hr, ipTempMover.Disable());
			END_IF
		END_WHILE
		
		IF CheckOk(hr) THEN 
			nSeqDisabling := 180;
		ELSE
			nSeqDisabling := 1000 + nSeqDisabling;
		END_IF			
		
		
	180: // Disabling movers
		THIS^.fbMovers.ResetIterator();
		WHILE THIS^.fbMovers.HasNextObject() DO
			IF ToMover(THIS^.fbMovers.GetNextObject(),ipTempMover) THEN
				hr := GetMostSignificant(hr, ipTempMover.Feedback.HR);
			END_IF
		END_WHILE
		
		IF CheckOk(hr) THEN 
			nSeqDisabling := 200;
		ELSIF FAILED(hr) THEN
			nSeqDisabling := 1000 + nSeqDisabling;
		END_IF		

		
	200: // Wait 1 second according to documentation
		fbTimeWait.IN := TRUE;
		fbTimeWait.PT := T#1S;	
		fbTimeWait();
		
		IF fbTimeWait.Q THEN
			fbTimeWait.IN := FALSE;
			fbTimeWait();
			nSeqDisabling := SEQ_DONE;
		END_IF
	
		
   SEQ_DONE: //Done
   		Disabling := S_OK;

		
	1000..1999://Error
		hr := GetMostSignificant(hrLastCycle, E_FAIL);	
END_CASE


//store last information
hrLastCycle := hr;


// Propagate error
IF FAILED(hr) THEN
	Disabling := hr;
END_IF
END_METHOD

METHOD Enable : CHALET_BaseComponents.I_CH_Feedback
VAR_INPUT
END_VAR
IF NOT THIS^.fbFeedback.Done THEN
	//Error active/not ready
	THIS^.fbFeedback.LastCommandAccepted 	:= FALSE;

ELSIF nSeqEnabling <> 0 THEN
	//System is partial or full enabled. Disable first.
	THIS^.fbFeedback.LastCommandAccepted 	:= FALSE;
ELSE
	
	THIS^.SuppressAllDynamicsChanges := FALSE;	

	THIS^.nSeqDisabling 	:= 0;
	THIS^.nSeqEnabling 		:= 1;
	
	THIS^.eActiveCommand 				:= CHALET_NC.E_NcAxisCommands.Enable;
	THIS^.fbFeedback.LastCommandAccepted:= TRUE;		
	THIS^.fbFeedback.Busy 				:= TRUE;	
END_IF

Enable := THIS^.fbFeedback;
END_METHOD

{attribute 'monitoring':='call'}
PROPERTY Enabled : BOOL
GET
Enabled := nSeqEnabling = SEQ_DONE;
END_GET
END_PROPERTY

METHOD PROTECTED Enabling : HRESULT
VAR
	hr : HRESULT;
	bWatchDogActive : BOOL;
	ipTempStation 	: I_XTS_Station;
	ipTempMover 	: I_XTS_Mover;
	nIdx 		: UDINT;
	nSupSeq : UINT;
END_VAR

VAR_INST
	fbTimeOutSeq 	: TON; 
	hrLastCycle 	: HRESULT;
	nlastState		: UINT;
	nModuleCount 	: UDINT;
	{attribute 'hide'}	
	fbTimeOutEnabling : FB_TcAlarm;
	{attribute 'hide'}	
	fbErrorEnabling : FB_TcAlarm;
END_VAR
Enabling := S_PENDING;
CASE nSeqEnabling OF
	0: // Idle
		Enabling := S_OK;

	1: // Check OP mode
		IF THIS^.ipEnvironment.UtilityEnvirement.XpuTcIo(1).GetOperationMode() = OperationMode.Normal THEN
			nSeqEnabling := 2; // Check 48V of all Module
		ELSE
			nSeqEnabling := 3; // in Simulation check of 48V not necessary
		END_IF
		
		
	2: // ToDo: check 48V of all Module?
		bWatchDogActive := TRUE;
		nModuleCount:= THIS^.ipEnvironment.UtilityEnvirement.XpuTcIo(1).PartTcIo(1).GetModuleCount();
		nSeqEnabling := 3;
		FOR nIdx := 1 TO nModuleCount DO
			IF THIS^.ipEnvironment.UtilityEnvirement.XpuTcIo(1).PartTcIo(1).ModuleTcIo(UDINT_TO_UINT(nIdx)).GetDCLinkVoltage() < 20 AND
			   THIS^.ipEnvironment.UtilityEnvirement.XpuTcIo(1).PartTcIo(1).ModuleTcIo(UDINT_TO_UINT(nIdx)).GetDCLinkVoltage() > 56 THEN	
				nSeqEnabling := 2;				     
			END_IF		
		END_FOR

		
	3: // ask for MoverId Detection Mode	
		bWatchDogActive := TRUE;
		IF Environment.UtilityEnvirement.XpuTcIo(1).GetMoverIdDetectionMode() = MoverIdDetectionMode.Standard THEN			
			nSeqEnabling := 10;
		ELSIF Environment.UtilityEnvirement.XpuTcIo(1).GetMoverIdDetectionMode() = MoverIdDetectionMode.Mover1 THEN
			nSeqEnabling := 5;
		ELSE // todo: MoverIdDetectionMode.MultipleMover1
			;
		END_IF
		

	5: // Trigger Mover ID dedection 
		bWatchDogActive := TRUE;
		IF NOT Environment.UtilityEnvirement.XpuTcIo(1).GetIsMoverIdDetectionActive() AND
		   NOT Environment.UtilityEnvirement.XpuTcIo(1).GetIsMoverIdDetectionValid() THEN
			// Set the Trigger for ID detection
			Environment.UtilityEnvirement.XpuTcIo(1).TriggerMoverIdDetection();
		ELSIF Environment.UtilityEnvirement.XpuTcIo(1).GetIsMoverIdDetectionValid() THEN
			// successful
			nSeqEnabling := 10;
		ELSIF Environment.UtilityEnvirement.XpuTcIo(1).GetHasMoverIdDetectionError() THEN
			// error
			nSeqEnabling := 1000 + nSeqEnabling;
		ELSE 
			; // wait for valid or error					
		END_IF
		
	
	10: // Reset movers
		bWatchDogActive := TRUE;
		THIS^.fbMovers.ResetIterator();
		WHILE THIS^.fbMovers.HasNextObject() DO
			IF ToMover(THIS^.fbMovers.GetNextObject(), ipTempMover) THEN
				hr := GetMostSignificant(hr, ipTempMover.Reset());
			END_IF
		END_WHILE
		
		IF CheckOk(hr) THEN 
			nSeqEnabling := 20;
		ELSE
			nSeqEnabling := 1000 + nSeqEnabling;
		END_IF
		
		
	20: // Resetting movers
		bWatchDogActive := TRUE;
		THIS^.fbMovers.ResetIterator();
		WHILE THIS^.fbMovers.HasNextObject() DO
			IF toMover(THIS^.fbMovers.GetNextObject(), ipTempMover) THEN
				hr := GetMostSignificant(hr, ipTempMover.Feedback.HR);
			END_IF
		END_WHILE
		
		IF CheckOk(hr) THEN 
			nSeqEnabling := 100;
		ELSIF FAILED(hr) THEN
			nSeqEnabling := 1000 + nSeqEnabling;
		END_IF	
		

	100..199: // Config Station
	(* All stations are always active to the same step to ensure that all data is available in the next step.
	   The following 100 steps are defined in the station. This makes overwriting easier *)
	   
		bWatchDogActive := TRUE;
		nSupSeq := nSeqEnabling - 100;
		THIS^.fbStations.ResetIterator();
		WHILE THIS^.fbStations.HasNextObject() DO
			IF ToStation(THIS^.fbStations.GetNextObject(),ipTempStation) THEN
				//Call this Methode whith seq 0->99, and wait each step until S_OK is returned. Call agaiin on S_Pending
				hr := GetMostSignificant(hr, ipTempStation.Configure(nSupSeq));
			END_IF
		END_WHILE	   
	   THIS^.fbStations.RestoreIterator();
	   
	   	IF CheckOk(hr) AND nSupSeq >= 99 THEN
			//All steps done 
			nSeqEnabling := 210;
		ELSIF FAILED(hr) THEN
			//Error
			nSeqEnabling := 1000 + nSeqEnabling;
		ELSIF CheckOk(hr) THEN 	 
			//active step is done, continous with next
			nSeqEnabling := nSeqEnabling + 1;
		END_IF	

	
	210: // Enable movers
		bWatchDogActive := TRUE;
		THIS^.fbMovers.ResetIterator();
		WHILE THIS^.fbMovers.HasNextObject() DO
			IF ToMover(THIS^.fbMovers.GetNextObject(),ipTempMover) THEN
				hr := GetMostSignificant(hr, ipTempMover.Enable());				 
			END_IF
		END_WHILE
		
		IF CheckOk(hr) THEN 
			nSeqEnabling := 220;
		ELSE
			nSeqEnabling := 1000 + nSeqEnabling;
		END_IF	
		

	220: // Enabling movers
		bWatchDogActive := TRUE;
		THIS^.fbMovers.ResetIterator();
		WHILE THIS^.fbMovers.HasNextObject() DO
			IF ToMover(THIS^.fbMovers.GetNextObject(),ipTempMover) THEN
				hr := GetMostSignificant(hr, ipTempMover.Feedback.HR);	
			END_IF
		END_WHILE
		
		IF CheckOk(hr) THEN 
			nSeqEnabling := 230;
		ELSIF FAILED(hr) THEN
			nSeqEnabling := 1000 + nSeqEnabling;
		END_IF
		
		
	230: // Add movers to group
		bWatchDogActive := TRUE;
		hr := THIS^.ipGroup.AddAxisListToGroup(fbMovers);
		
		IF CheckOk(hr) THEN 
			nSeqEnabling := 240;
		ELSE
			nSeqEnabling := 1000 + nSeqEnabling;
		END_IF	
		

	240: // Adding mover to group
		bWatchDogActive := TRUE;
		hr := THIS^.ipGroup.AddingAxisToGroup();
		
		IF CheckOk(hr) THEN 
			nSeqEnabling := 250;
		ELSIF FAILED(hr) THEN
			nSeqEnabling := 1000 + nSeqEnabling;
		END_IF		
		
		
	250: // Enable group
		bWatchDogActive := TRUE;
		hr :=THIS^.ipGroup.Enable();
		
		IF CheckOk(hr) THEN 
			nSeqEnabling := 260;
		ELSE
			nSeqEnabling := 1000 + nSeqEnabling;
		END_IF	
		
		
	260: // Enabling group
		bWatchDogActive := TRUE;
		hr := THIS^.ipGroup.HR;
		
		IF THIS^.ipGroup.GroupEnabled THEN 
			nSeqEnabling := SEQ_DONE;
		ELSIF FAILED(hr) THEN
			nSeqEnabling := 1000 + nSeqEnabling;
		END_IF	
		
		
	SEQ_DONE: // Done
		Enabling := S_OK;


	1000..1999://Error
		hr := GetMostSignificant(hrLastCycle, E_FAIL);
		//Only rais if timeout is not active
		IF NOT fbErrorEnabling.bRaised AND NOT fbTimeOutEnabling.bRaised THEN 
			fbErrorEnabling.CreateEx(stEventEntry:=TC_EVENTS.CHALET_Base_Events.ErrorEnabling, ipSourceInfo := THIS^.fbSourceInfo, bWithConfirmation := FALSE);
			fbErrorEnabling.ipArguments.AddUInt(nSeqEnabling-1000);
			fbErrorEnabling.Raise(0);
		END_IF
END_CASE


//Timeout after to long stay in one of the following seq.
fbTimeOutSeq.IN := (nlastState = nSeqEnabling) AND bWatchDogActive;
fbTimeOutSeq.PT := T#10S;
fbTimeOutSeq();
nlastState := nSeqEnabling;

IF fbTimeOutSeq.Q THEN
	IF NOT fbTimeOutEnabling.bRaised THEN 
		fbTimeOutEnabling.CreateEx(stEventEntry:=TC_EVENTS.CHALET_Base_Events.TimeOutEnabling, ipSourceInfo := THIS^.fbSourceInfo, bWithConfirmation := FALSE);
		fbTimeOutEnabling.ipArguments.AddUInt(nSeqEnabling);
		fbTimeOutEnabling.Raise(0);
	END_IF
	//next seq is error
	nSeqEnabling := 1000 + nSeqEnabling;
END_IF

//Clear Tc3-Eventlogger alarm 
IF nSeqEnabling <= SEQ_DONE THEN
	fbTimeOutEnabling.Clear(0,0);
	fbErrorEnabling.Clear(0,0);
END_IF


//store last information
hrLastCycle := hr;

// Propagate error
IF FAILED(hr) THEN
	Enabling := hr;
END_IF
END_METHOD

{attribute 'monitoring':='call'}
PROPERTY Environment : I_XTS_Environment
GET
Environment := THIS^.ipEnvironment;
END_GET
END_PROPERTY

{attribute 'monitoring':='call'}
PROPERTY Feedback : CHALET_BaseComponents.I_CH_Feedback
GET
Feedback := THIS^.fbFeedback;
END_GET
END_PROPERTY

METHOD getMoverInFront : I_Xts_Mover
VAR_INPUT
	ipMover	: I_Xts_Mover;
END_VAR

VAR
	fPosOnTrack			: LREAL;
	ipTempMover 		: I_XTS_Mover;
	fTempPosOnTrack		: LREAL;
	fTempDistBetween 	: LREAL;
	
	fFoundDistBetween : LREAL := CHALET_BaseComponents.GVL_Datatypes.cMaxLreal;
	ipFoundMover	: I_Xts_Mover;
END_VAR
//use NcToPlc.ModuloActPos because iMover.PositionOnTrack is not ready during init
//get an copy of the mover list 
//fbTempListOfMovers.Duplicate(THIS^.fbMovers);


// get postion of myself
fPosOnTrack := ipMover.getAxisRef.NcToPlc.ModuloActPos;

// go through the list and search the mover in front
THIS^.fbMovers.ResetIterator();
WHILE THIS^.fbMovers.HasNextObject() DO
	IF ToMover(THIS^.fbMovers.GetNextObject(), ipTempMover) THEN
		// if Mover is myself, skipp
		IF ipTempMover <> ipMover THEN
			// calc distance to Mover in positive direction
			fTempDistBetween := F_GetDistToPosModulo(fActualPosition := fPosOnTrack, fTargedPosition := ipTempMover.getAxisRef.NcToPlc.ModuloActPos, fModulo := TrackLength);
	
	
			// check if Mover is closer then last one
			IF fFoundDistBetween > fTempDistBetween THEN 
				fFoundDistBetween := fTempDistBetween;
				ipFoundMover := ipTempMover;
			END_IF
		END_IF
	END_IF
END_WHILE

getMoverInFront := ipFoundMover;
END_METHOD

METHOD getStationInFront : I_XTS_Station
VAR_INPUT
	ipStation	: I_XTS_Station;
END_VAR
VAR
	fPosOnTrack			: LREAL;
	
	ipTempStation 		: I_XTS_Station;
	fTempPosOnTrack		: LREAL;
	fTempDistBetween 	: LREAL;
	
	fFoundDistBetween 	: LREAL := CHALET_BaseComponents.GVL_Datatypes.cMaxLreal;
	ipFoundStation		: I_XTS_Station;
END_VAR
// get postion of myself
fPosOnTrack := ipStation.PositionOnTrack;

// go through the list and search the station in front
THIS^.fbStations.ResetIterator();
WHILE THIS^.fbStations.HasNextObject() DO
	IF ToStation(THIS^.fbStations.GetNextObject(), ipTempStation) THEN
		// calc distance to Station
		fTempDistBetween := ipTempStation.PositionOnTrack - fPosOnTrack;		
		
		// if Station is behinde me or it is myself -> add Modulo
		IF fTempDistBetween <= 0 AND THIS^.Environment.TrackIsRing THEN 
			fTempDistBetween := fTempDistBetween + TrackLength;			
		END_IF

		// check if Station is closer then last one
		IF fFoundDistBetween > fTempDistBetween THEN 
			fFoundDistBetween := fTempDistBetween;
			ipFoundStation := ipTempStation;
		END_IF
		
	END_IF
END_WHILE

getStationInFront := ipFoundStation;
END_METHOD

METHOD Initialize : HRESULT
VAR
	hr : HRESULT;
END_VAR


VAR_INST
	//This error cannot be reset. Requires a reset cold
	{attribute 'hide'}	
	fbInitError : FB_TcAlarm;
END_VAR
//Set to busy on first call
IF THIS^.eActiveCommand <> CHALET_NC.E_NcAxisCommands.Initialize THEN
	THIS^.eActiveCommand 					:= CHALET_NC.E_NcAxisCommands.Initialize;
	THIS^.fbFeedback.LastCommandAccepted	:= TRUE;		
	THIS^.fbFeedback.Busy 					:= TRUE;
END_IF


//Check Error during FB_Init
IF THIS^.bErrorDuringFbInit THEN
	IF NOT fbInitError.bRaised THEN 
		//This error cannot be reset. Requires a reset cold
		fbInitError.CreateEx(stEventEntry:=TC_EVENTS.CHALET_Base_Events.ErrorFBinit, ipSourceInfo := THIS^.fbSourceInfo, bWithConfirmation := FALSE);
		fbInitError.Raise(0);
	END_IF
	Initialize:= E_FAIL;
	THIS^.fbFeedback.HR := Initialize;
	RETURN;
END_IF	

//Check if Envirement and Group is existing
IF THIS^.ipGroup = 0 THEN
	IF NOT fbInitError.bRaised THEN 
		//This error cannot be reset. Requires a reset cold
		fbInitError.CreateEx(stEventEntry:=TC_EVENTS.CHALET_XTS_Events.MissingGroupe, ipSourceInfo := THIS^.fbSourceInfo, bWithConfirmation := FALSE);
		fbInitError.Raise(0);
	END_IF
	Initialize:= E_FAIL;
	THIS^.fbFeedback.HR := Initialize;
	RETURN;
END_IF	

//Check if Envirement and Group is existing
IF THIS^.ipEnvironment = 0 THEN
	IF NOT fbInitError.bRaised THEN 
		//This error cannot be reset. Requires a reset cold
		fbInitError.CreateEx(stEventEntry:=TC_EVENTS.CHALET_XTS_Events.MissingEnvironment, ipSourceInfo := THIS^.fbSourceInfo, bWithConfirmation := FALSE);
		fbInitError.Raise(0);
	END_IF
	Initialize:= E_FAIL;
	THIS^.fbFeedback.HR := Initialize;
	RETURN;
END_IF	




//Init Envirement. This includes XTS_Utility
hr := GetMostSignificant(hr, ipEnvironment.Initialize());	

//Init envirement first to get access to XTS_Utility
IF THIS^.ipEnvironment.UtilityEnvirement.P_IsInitialized THEN
	hr := GetMostSignificant(hr, fbMovers.Initialize());	
	hr := GetMostSignificant(hr, ipGroup.Initialize());	
	hr := GetMostSignificant(hr, fbStations.Initialize());	
	
	//Init Zone and Trigger only if main components are initialized
	IF hr = S_OK THEN
		hr := GetMostSignificant(hr, fbZones.Initialize());	
		hr := GetMostSignificant(hr, fbTriggers.Initialize());	
	END_IF
ELSE
	hr := GetMostSignificant(hr, S_PENDING);
END_IF	


THIS^.bInitDone := (hr = S_OK);

Initialize:= hr;

THIS^.fbFeedback.HR := Initialize;
END_METHOD

{attribute 'monitoring':='call'}
PROPERTY Initialized : BOOL
GET
Initialized := bInitDone;
END_GET
END_PROPERTY

METHOD LinkEnvironment : HRESULT
VAR_INPUT
	ipEnvironment	: CHALET_BaseComponents.I_CH_Object;
END_VAR

VAR
	ipXtsEnvironment : I_Xts_Environment;
END_VAR
IF ipEnvironment <> 0 AND_THEN __QUERYINTERFACE(ipEnvironment, ipXtsEnvironment) THEN
	THIS^.ipEnvironment := ipXtsEnvironment;
	LinkEnvironment := S_OK;
ELSE
	LinkEnvironment := E_FAIL;
	THIS^.bErrorDuringFbInit := TRUE;
END_IF
END_METHOD

METHOD LinkGroup : HRESULT
VAR_INPUT
	ipGroup	: CHALET_BaseComponents.I_CH_Object;
END_VAR

VAR
	ipXtsGroup : I_XTS_Group;
END_VAR
IF ipGroup <> 0 AND_THEN __QUERYINTERFACE(ipGroup, ipXtsGroup) THEN
	THIS^.ipGroup := ipXtsGroup;
	LinkGroup := S_OK;
ELSE
	LinkGroup := E_FAIL;
	THIS^.bErrorDuringFbInit := TRUE;
END_IF
END_METHOD

{attribute 'monitoring':='call'}
PROPERTY Movers : CHALET_BaseComponents.I_CH_LIST
GET
Movers := THIS^.fbMovers;
END_GET
END_PROPERTY

METHOD RegisterMover : HRESULT
VAR_INPUT
	ipMover	: CHALET_BaseComponents.I_CH_Object;
END_VAR

VAR
	ipXtsMover : I_XTS_Mover;
END_VAR
IF ipMover = 0 THEN
	//Invalide interface	
	THIS^.bErrorDuringFbInit := TRUE;
	RegisterMover := E_FAIL;
	
ELSIF NOT __QUERYINTERFACE(ipMover, ipXtsMover) THEN
	//The required interface is missing
	THIS^.bErrorDuringFbInit := TRUE;
	RegisterMover := E_FAIL;
	
ELSIF THIS^.fbMovers.IsFull THEN
	//List is full
	THIS^.bErrorDuringFbInit := TRUE;
	RegisterMover := E_FAIL;
	
ELSIF THIS^.bInitDone THEN
	//To late. System is initilized
	THIS^.bErrorDuringFbInit := TRUE;
	RegisterMover := E_FAIL;
	
ELSE
	
	THIS^.fbMovers.AddObject(ipMover);
END_IF
END_METHOD

METHOD RegisterStation : HRESULT
VAR_INPUT
	ipStation	: CHALET_BaseComponents.I_CH_Object;
END_VAR

VAR
	ipXtsStation : I_XTS_Station;
END_VAR
IF ipStation = 0 THEN
	//Invalide interface	
	THIS^.bErrorDuringFbInit := TRUE;
	RegisterStation := E_FAIL;
	
ELSIF NOT __QUERYINTERFACE(ipStation, ipXtsStation) THEN
	//The required interface is missing
	THIS^.bErrorDuringFbInit := TRUE;
	RegisterStation := E_FAIL;
	
ELSIF THIS^.fbStations.IsFull THEN
	//List is full
	THIS^.bErrorDuringFbInit := TRUE;
	RegisterStation := E_FAIL;
	
ELSIF THIS^.bInitDone THEN
	//To late. System is initilized
	THIS^.bErrorDuringFbInit := TRUE;
	RegisterStation := E_FAIL;
		
ELSE
	
	THIS^.fbStations.AddObject(ipStation);
END_IF
END_METHOD

METHOD RegisterTrigger : HRESULT
VAR_INPUT
	ipTrigger	: CHALET_BaseComponents.I_CH_Object;
END_VAR
VAR
	ipXtsTrigger : I_XTS_Trigger;
END_VAR
IF ipTrigger = 0 THEN
	//Invalide interface	
	THIS^.bErrorDuringFbInit := TRUE;
	RegisterTrigger := E_FAIL;
	
ELSIF NOT __QUERYINTERFACE(ipTrigger, ipXtsTrigger) THEN
	//The required interface is missing
	THIS^.bErrorDuringFbInit := TRUE;
	RegisterTrigger := E_FAIL;
	
ELSIF THIS^.fbTriggers.IsFull THEN
	//List is full
	THIS^.bErrorDuringFbInit := TRUE;
	RegisterTrigger := E_FAIL;
	
ELSIF THIS^.bInitDone THEN
	//To late. System is initilized
	THIS^.bErrorDuringFbInit := TRUE;
	RegisterTrigger := E_FAIL;
		
ELSE
	
	THIS^.fbTriggers.AddObject(ipTrigger);
END_IF
END_METHOD

METHOD RegisterZone : HRESULT
VAR_INPUT
	ipZone	: CHALET_BaseComponents.I_CH_Object;
END_VAR
VAR
	ipXtsZone : I_XTS_Zone;
END_VAR
IF ipZone = 0 THEN
	//Invalide interface	
	THIS^.bErrorDuringFbInit := TRUE;
	RegisterZone := E_FAIL;

ELSIF NOT __QUERYINTERFACE(ipZone, ipXtsZone) THEN
	//The required interface is missing
	THIS^.bErrorDuringFbInit := TRUE;
	RegisterZone := E_FAIL;
	
ELSIF THIS^.fbZones.IsFull THEN
	//List is full
	THIS^.bErrorDuringFbInit := TRUE;
	RegisterZone := E_FAIL;
	
ELSIF THIS^.bInitDone THEN
	//To late. System is initilized
	THIS^.bErrorDuringFbInit := TRUE;
	RegisterZone := E_FAIL;
		
ELSE
	
	THIS^.fbZones.AddObject(ipZone);	
END_IF
END_METHOD

METHOD Reset : HRESULT
VAR
	hr : HRESULT;
	bOk : BOOL := TRUE;
	ipTempMover : I_XTS_Mover;
END_VAR
// Reset movers
THIS^.fbMovers.ResetIterator();
WHILE THIS^.fbMovers.HasNextObject() DO
	IF ToMover(THIS^.fbMovers.GetNextObject(),ipTempMover) THEN
		hr := GetMostSignificant(hr, ipTempMover.Reset());
	END_IF
END_WHILE
	
// Reset groupe	
IF THIS^.ipGroup <> 0 THEN
	GetMostSignificant(hr, THIS^.ipGroup.Reset());
END_IF

Reset := hr;
END_METHOD

METHOD Station : I_XTS_Station_PLC
VAR_INPUT
	sLUID	: STRING;
END_VAR
//IF no station was found, INTERFACE is 0 -> can generate fatal error
__QUERYINTERFACE(THIS^.fbStations.FindLUID(sLUID),Station);
END_METHOD

{attribute 'monitoring':='call'}
PROPERTY Stations : CHALET_BaseComponents.I_CH_LIST
GET
Stations := THIS^.fbStations;
END_GET
END_PROPERTY

//Suppress to change the dynamic(Gap+velocity) of passing movers in all stations. This is usefull in startup
PROPERTY SuppressAllDynamicsChanges : BOOL
SET
VAR
	ipTempStationPlc : I_XTS_Station_PLC;
END_VAR
// go through the list and write request to it
THIS^.fbStations.ResetIterator();
WHILE THIS^.fbStations.HasNextObject() DO
	IF ToStation_PLC(THIS^.fbStations.GetNextObject(), ipTempStationPlc) THEN
		ipTempStationPlc.SuppressDynamicsChange := SuppressAllDynamicsChanges;
	END_IF
END_WHILE
END_SET
END_PROPERTY

{attribute 'monitoring':='call'}
PROPERTY TrackLength : LREAL
GET
TrackLength := THIS^.ipEnvironment.TrackLength;
END_GET
END_PROPERTY

{attribute 'monitoring':='call'}
PROPERTY Triggers : CHALET_BaseComponents.I_CH_LIST
GET
Triggers := THIS^.fbTriggers;
END_GET
END_PROPERTY

METHOD Update : HRESULT
VAR_INPUT
END_VAR
VAR
	hr : HRESULT;
END_VAR
//Force to do an init at beginn
IF NOT THIS^.Initialized THEN
	THIS^.Initialize();
	RETURN;
END_IF

hr := S_OK;

hr := GetMostSignificant(hr, THIS^.Enabling());	
hr := GetMostSignificant(hr, THIS^.Disabling());	




// ********************** Set feedback depending on active command *******************************
IF THIS^.eActiveCommand <> E_NcAxisCommands.None THEN
	fbFeedback.ActiveCommand 	:= TO_STRING(THIS^.eActiveCommand);	
END_IF

CASE THIS^.eActiveCommand OF
	E_NcAxisCommands.None: 
		;

	E_NcAxisCommands.Initialize:
		fbFeedback.Busy 		:= NOT THIS^.bInitDone;
		fbFeedback.Done 		:= THIS^.bInitDone;
		fbFeedback.ErrorId 		:= 0;
		
	E_NcAxisCommands.Enable:
		fbFeedback.Busy 		:= nSeqEnabling > 0;
		fbFeedback.Done 		:= THIS^.Enabled;
		IF nSeqEnabling > 1000 THEN
			fbFeedback.ErrorId 		:= nSeqEnabling;
		END_IF
		
	E_NcAxisCommands.Disable:
		fbFeedback.Busy 		:= nSeqDisabling > 0;
		fbFeedback.Done 		:= THIS^.Disabled;
		IF nSeqDisabling > 1000 THEN
			fbFeedback.ErrorId 		:= nSeqDisabling;
		END_IF
		


	ELSE//External command in subclass
		;
END_CASE


// **********************  Stop to execute commands on .done or .error ***************************
IF fbFeedback.Done OR THIS^.fbFeedback.Error THEN
	eActiveCommand 				:= E_NcAxisCommands.None;
END_IF







hr := GetMostSignificant(hr, THIS^.fbMovers.Update());	
hr := GetMostSignificant(hr, THIS^.fbStations.Update());	
hr := GetMostSignificant(hr, THIS^.fbZones.Update());	
hr := GetMostSignificant(hr, THIS^.fbTriggers.Update());	


hr := GetMostSignificant(hr, THIS^.ipGroup.Update());	
hr := GetMostSignificant(hr, THIS^.ipEnvironment.Update());	

Update:= hr;
END_METHOD

{attribute 'monitoring':='call'}
PROPERTY Zones : CHALET_BaseComponents.I_CH_LIST
GET
Zones := THIS^.fbZones;
END_GET
END_PROPERTY

END_FUNCTION_BLOCK
